{attribute 'qualified_only'}
VAR_GLOBAL
	axis : AXIS_REF;
	pBEnableMotor : BOOL;
	pbDisableMotor : BOOL;
	motorIsEnabled : BOOL;
	motorIsReallyEnabled : BOOL;
	pBJog : BOOL;
	jogError: BOOL;
	pBMoveVelocity : BOOL;
	pBHalt : BOOL;
END_VAR

(* stored: Version 1.1.0.1, ProductVersion 3.1.4024.12
   GVL GVL: Id {655dbc17-70e0-4cbd-8edb-f6745b719644} *)
